(* IEC 61131-3 sources: POC_CAu/, 3 files *)

(* ---- Main 2.0.ST ---- *)
VAR_GLOBAL

//OUTPUT
glob_Pist1 at %Y33.1:BOOL;                                             //pist pod otvorem na vlozeni obrobku
glob_Pist2 at %Y33.0:BOOL;                                             //pist pro lisovani obrobku
glob_Kompresor at %Y33.2:BOOL;                                         //kompresor
glob_MotorStolu at %Y32.5:BOOL;                                        //motor otocneho stolu
glob_DvoucinnyPist1 at %Y32.6:BOOL;                                    //vysunuti dvoucinneho pistu nad dopravnikem
glob_DvoucinnyPist2 at %Y32.7:BOOL;                                    //zasunuti dvoucinneho pistu nad dopravnikem
glob_MotorDopravniku at %Y32.4:BOOL;

//INPUT
glob_Dioda1 at %X100.6:BOOL;                                           //svetelna zavora pod otvorem na vlozeni obrobku
glob_Dioda2 at %X100.0:BOOL;                                           //svetelna zavora na dopravniku
glob_Start_Stop at %X100.7:BOOL;                                       //tlacitko start-stop
glob_TrigStolu at %X100.5:BOOL;                                        //tlacitko, ktere stiskava otoc. stul
glob_tlacitkoPist2 at  %X100.4:BOOL;                                   //tlacitko pod lisem
glob_TlacitkoDopravniku at %X100.1:BOOL;                               //tlacitko u dopravniku

pocetVyrobku: UDINT := 0;
pomSTTrig: USINT := 0;
pomocnaStav:USINT;

glob_KillSwitch:BOOL;

END_VAR

///////////////////////////////////////////////////////////////////////////////////////////////////////////////////////////////////////////////////////////////////////////////////////////////////////

FUNCTION_BLOCK fb_VychoziStav                                          //pocatecni funkce pro nastveni stolu na vychozi pozici

VAR_INPUT
talcitko:BOOL;
END_VAR

VAR_OUTPUT
vystup:BOOL;
END_VAR

VAR
stisknuto:BOOL;
nabezna:R_TRIG;
END_VAR

nabezna(CLK := talcitko,Q => stisknuto);

glob_KillSwitch := glob_KillSwitch XOR stisknuto;

IF glob_TrigStolu = FALSE AND glob_KillSwitch = TRUE THEN
vystup := TRUE;
ELSIF glob_TrigStolu = TRUE THEN
vystup := FALSE;
END_IF;

END_FUNCTION_BLOCK
///////////////////////////////////////////////////////////////////////////////////////////////////////////////////////////////////////////////////////////////////////////////////////////////////////

FUNCTION_BLOCK fb_VypnouLinku                                           //funkce pro vypinani cele linky

VAR_INPUT
talcitko:BOOL;
END_VAR

VAR_OUTPUT
vystup:BOOL;
END_VAR

VAR
stisknuto:BOOL;
nabezna:R_TRIG;
END_VAR

nabezna(CLK := talcitko,Q => stisknuto);

vystup := vystup XOR stisknuto;

IF vystup = FALSE THEN
pomocnaStav:=4;                                                        //obrazuje na display PLC "Pozastaveno"
END_IF;

END_FUNCTION_BLOCK
///////////////////////////////////////////////////////////////////////////////////////////////////////////////////////////////////////////////////////////////////////////////////////////////////////

FUNCTION_BLOCK fb_PozicePist1

VAR_INPUT
dioda1:BOOL;
dioda2:BOOL;
END_VAR

VAR_OUTPUT
vystup1:BOOL;
vystup2:BOOL;
vystup3:BOOL;
END_VAR

VAR
zapnuto:BOOL;
zpozdovac:TON;
END_VAR

zpozdovac1(IN := glob_KillSwitch AND glob_TrigStolu AND NOT dioda1 AND dioda2,PT := T#2s,Q => zapnuto);
vystup1 := zapnuto;
vystup2 := zapnuto;
zpozdovac2(IN := glob_KillSwitch AND dioda1 AND dioda2 AND NOT glob_TlacitkoPist2,PT := T#3s,Q => vystup3);

END_FUNCTION_BLOCK
///////////////////////////////////////////////////////////////////////////////////////////////////////////////////////////////////////////////////////////////////////////////////////////////////////

FUNCTION_BLOCK fb_PoziceLis

VAR_INPUT
tlacitko:BOOL;
END_VAR

VAR_OUTPUT
vystup1:BOOL;
vystup2:BOOL;
vystup3:BOOL;
END_VAR

VAR
zapnuto:BOOL;
zpozdovac:TON;
END_VAR

IF tlacitko = TRUE THEN
zpozdovac(IN := glob_KillSwitch AND glob_TlacitkoPist2,PT := T#5s,Q => zapnuto);
vystup1 := zapnuto;
vystup2 := zapnuto;
vystup3 := zapnuto;
END_IF;

END_FUNCTION_BLOCK
///////////////////////////////////////////////////////////////////////////////////////////////////////////////////////////////////////////////////////////////////////////////////////////////////////

fb_PoziceDopravnik

VAR_INPUT
pist:BOOL;
END_VAR

VAR_OUTPUT
vystup:BOOL;
END_VAR

VAR
vypnut,zapnuto:BOOL;
zpozdovac:TON;
sestupna:F_TRIG;
nabezna:R_TRIG;
END_VAR

sestupna(CLK := pist,Q => vypnut);

IF vypnut = TRUE THEN
glob_MotorStolu := TRUE;
ELSIF glob_TlacitkoDopravniku = TRUE THEN
glob_MotorStolu := FALSE;
END_IF;

zpozdovac(IN := glob_KillSwitch AND glob_TlacitkoDopravniku AND glob_Dioda2,PT := T#1s,Q => vystup);

nabezna(CLK := vystup,Q => zapnuto);

IF zapnuto AND glob_Dioda2 THEN
glob_Kompresor := FALSE;
glob_MotorDopravniku := TRUE;
ELSIF glob_KillSwitch AND NOT glob_Dioda2 THEN
glob_MotorDopravniku := FALSE;
//pocetVyrobku:= pocetVyrobku + 1;
pomocnaStav:=2;                                                        //zobrazuje na display PLC "Odeberte obrobek"
END_IF;

END_FUNCTION_BLOCK
///////////////////////////////////////////////////////////////////////////////////////////////////////////////////////////////////////////////////////////////////////////////////////////////////////

PROGRAM Main

fb_VychoziStav(glob_Start_Stop := tlacitko,vystup := glob_MotorStolu);
fb_VypnouLinku(glob_Start_Stop := tlacitko,vystup := glob_KillSwitch);
fb_PozicePist1(glob_Dioda1 := dioda1,glob_Dioda2 := dioda2,glob_Kompresor := vystup1,glob_Pist1 := vystup2,glob_MotorStolu := vystup3);
fb_PoziceLis(glob_TlacitkoPist2 := tlacitko,glob_Kompresor := vystup1,glob_Pist2 := vystup2,glob_DvoucinnyPist1 := vystup3);
fb_PoziceDopravnik(glob_Pist2 := pist,);

END_PROGRAM

(* ---- prgMain.ST ---- *)
VAR_GLOBAL

//OUTPUT
glob_Pist1 at %Y33.1:BOOL;                                             //pist pod otvorem na vlozeni obrobku
glob_Pist2 at %Y33.0:BOOL;                                             //pist pro lisovani obrobku
glob_Kompresor at %Y33.2:BOOL;                                         //kompresor
glob_MotorStolu at %Y32.5:BOOL;                                        //motor otocneho stolu
glob_DvojcinnyPist1 at %Y32.6:BOOL;                                    //vysunuti dvoucinneho pistu nad dopravnikem
glob_DvojcinnyPist2 at %Y32.7:BOOL;                                    //zasunuti dvoucinneho pistu nad dopravnikem
glob_MotorDopravniku at %Y32.4:BOOL;

//INPUT
glob_Dioda1 at %X100.6:BOOL;                                           //svetelna zavora pod otvorem na vlozeni obrobku
glob_Dioda2 at %X100.0:BOOL;                                           //svetelna zavora na dopravniku
glob_Start_Stop at %X100.7:BOOL;                                       //tlacitko start-stop
glob_TrigStolu at %X100.5:BOOL;                                        //tlacitko, ktere stiskava otoc. stul
glob_tlacitkoPist2 at  %X100.4:BOOL;                                   //tlacitko pod lisem
glob_TlacitkoDopravniku at %X100.1:BOOL;                               //tlacitko u dopravniku

pocetVyrobku: UDINT := 0;
pomocnaStav:USINT;

glob_KillSwitch:BOOL;

END_VAR

///////////////////////////////////////////////////////////////////////////////////////////////////////////////////////////////////////////////////////////////////////////////////////////////////////

FUNCTION_BLOCK fb_VychoziStav

VAR_INPUT
tlacitko:BOOL;
END_VAR

VAR
stisknuto:BOOL;
nabezna:R_TRIG;
END_VAR

nabezna(CLK := tlacitko,Q => stisknuto);
glob_KillSwitch := glob_KillSwitch XOR stisknuto;

IF stisknuto = TRUE THEN
 pomocnaStav:=0;
END_IF;

IF NOT glob_TrigStolu AND glob_KillSwitch THEN
 glob_MotorStolu := TRUE;
ELSIF glob_TrigStolu AND glob_KillSwitch THEN
 glob_MotorStolu := FALSE;
END_IF;

IF glob_KillSwitch = FALSE THEN
 pomocnaStav:=2;
END_IF;

END_FUNCTION_BLOCK
///////////////////////////////////////////////////////////////////////////////////////////////////////////////////////////////////////////////////////////////////////////////////////////////////////

FUNCTION_BLOCK fb_PozicePist1

VAR_INPUT
dioda1:BOOL;
END_VAR

VAR
zapnuto1,zapnuto2,probehlo,pom:BOOL;
zpozdovac1,zpozdovac2:TON;
sestup:F_TRIG;
END_VAR

IF NOT dioda1 THEN
 pomocnaStav:=4;
END_IF;

zpozdovac1(IN := NOT dioda1,PT := T#2s0ms,Q => zapnuto1);

IF zapnuto1 = TRUE THEN
 glob_Kompresor := TRUE;
 glob_Pist1 := TRUE;
 pomocnaStav:=3;
ELSE
 glob_Kompresor := FALSE;
 glob_Pist1 := FALSE;
END_IF;

sestup(CLK := glob_Pist1,Q => probehlo);

if probehlo then;
   pom:=TRUE;
END_IF;

zpozdovac2(IN := pom,PT := T#3s0ms,Q => zapnuto2);

IF zapnuto2 and glob_KillSwitch THEN
   glob_MotorStolu := TRUE;
END_IF;

IF glob_tlacitkoPist2 = TRUE THEN
   glob_MotorStolu := FALSE;
   pom := FALSE;
END_IF;

END_FUNCTION_BLOCK
///////////////////////////////////////////////////////////////////////////////////////////////////////////////////////////////////////////////////////////////////////////////////////////////////////

FUNCTION_BLOCK fb_PoziceLis

VAR_INPUT
tlacitko:BOOL;
END_VAR

VAR
casovac:TP;
sestup:F_TRIG;
zapnuto,probehlo,pom:BOOL;
END_VAR

IF tlacitko = TRUE THEN
 casovac(IN := glob_KillSwitch AND glob_TlacitkoPist2,PT := T#5s0ms,Q => zapnuto);
 glob_Kompresor := zapnuto;
 glob_Pist2 := zapnuto;
 glob_DvojcinnyPist1 := zapnuto;
ELSE
 casovac(IN := FALSE);
END_IF;

sestup(CLK := glob_Pist2,Q => probehlo);

IF probehlo THEN;
 pom := TRUE;
END_IF;

IF pom AND glob_KillSwitch THEN
 glob_MotorStolu := TRUE;
END_IF;

IF glob_TlacitkoDopravniku = TRUE THEN
 glob_MotorStolu := FALSE;
 pom := FALSE;
END_IF;

END_FUNCTION_BLOCK
///////////////////////////////////////////////////////////////////////////////////////////////////////////////////////////////////////////////////////////////////////////////////////////////////////

FUNCTION_BLOCK fb_PoziceDopravnik

VAR_INPUT
tlacitko:BOOL;
END_VAR

VAR
zapnuto,konec,pom:BOOL;
zpozdovac:TON;
nabez:R_TRIG;
END_VAR

IF tlacitko = TRUE THEN
 glob_MotorDopravniku := TRUE;
END_IF;

zpozdovac(IN := glob_KillSwitch AND glob_MotorDopravniku AND glob_Dioda2,PT := T#1s,Q => zapnuto);

IF zapnuto = TRUE THEN
 glob_Kompresor := TRUE;
 glob_DvojcinnyPist2 := TRUE;
END_IF;

nabez(CLK:= NOT glob_Dioda2,Q => konec);

IF glob_Dioda2 = FALSE THEN
 glob_MotorDopravniku := FALSE;
END_IF;

IF konec = TRUE THEN
 pomocnaStav := 1;
 pocetVyrobku := pocetVyrobku + 1;
 pom := TRUE;
END_IF;

IF pom AND glob_Dioda2 THEN
 glob_KillSwitch := FALSE;
 pom := FALSE;
END_IF;

END_FUNCTION_BLOCK
///////////////////////////////////////////////////////////////////////////////////////////////////////////////////////////////////////////////////////////////////////////////////////////////////////

FUNCTION kill : BOOL
         glob_Pist1           :=0;
         glob_Pist2           :=0;
         glob_Kompresor       :=0;
         glob_MotorStolu      :=0;
         glob_DvojcinnyPist1  :=0;
         glob_DvojcinnyPist2  :=0;
         glob_MotorDopravniku :=0;
END_FUNCTION

VAR_GLOBAL
 fb_VS : fb_VychoziStav;
 fb_PP : fb_PozicePist1;
 fb_PL : fb_PoziceLis;
 fb_PD : fb_PoziceDopravnik;
END_VAR

PROGRAM prgMain
fb_VS(tlacitko := glob_Start_Stop);
IF glob_killswitch = TRUE THEN
 fb_PP(dioda1 := glob_Dioda1);
 fb_PL(tlacitko := glob_TlacitkoPist2);
 fb_PD(tlacitko := glob_TlacitkoDopravniku);
ELSE
 kill();
END_IF;

END_PROGRAM

(* ---- OLD_Main.ST ---- *)
VAR_GLOBAL

//OUTPUT
Pist1 at %Y33.1:BOOL;                                                  //pist pod otvorem na vlozeni obrobku
Pist2 at %Y33.0:BOOL;                                                  //pist pro lisovani obrobku
kompr at %Y33.2:BOOL;                                                  //kompresor
MotorStolu at %Y32.5:BOOL;                                             //motor otocneho stolu
DvoucinnyPist1 at %Y32.6:BOOL;                                         //vysunuti dvoucinneho pistu nad dopravnikem
DvoucinnyPist2 at %Y32.7:BOOL;                                         //zasunuti dvoucinneho pistu nad dopravnikem
MotorDopravniku at %Y32.4:BOOL;

//INPUT
Dioda1 at %X100.6:BOOL;                                                //svetelna zavora pod otvorem na vlozeni obrobku
Dioda2 at %X100.0:BOOL;                                                //svetelna zavora na dopravniku
StartStop at %X100.7:BOOL;                                             //tlacitko start-stop
tlacitkoStolu at %X100.5:BOOL;                                         //tlacitko, ktere stiskava otoc. stul
tlacitkoPist2 at  %X100.4:BOOL;                                        //tlacitko pod lisem
tlacitkoDopravniku at %X100.1:BOOL;                                    //tlacitko u dopravniku
pocetVyrobku: UDINT := 0;
pomSTTrig: USINT := 0;
pomocnaStav:USINT;
//prnt at %R1:array[0..79] of USINT;
END_VAR

PROGRAM prgMain

VAR

data:TIME;
nabez1,nebezHotovo:R_TRIG;
sestup1:F_TRIG;
SestupPist2:F_TRIG;
SestuptlacitkoDopravniku:F_TRIG;
Casovac1,Casovac2:TOF;
Zpozdovac1,Zpozdovac2,Zpozdovac3,Zpozdovac4:TON;
pomStart,pomPist1,pomPist2,pomMotorS,pom1,pom3,pom5,pom6,pom7,pom9,pom10,pom11,pom12,pom13,pom14,pom15,pom16,pom17,pom18,pomZap,pomses,pomStop,pomPist1kon,pomZpozdeni,pomHotovo,pomHotovo2,pomHotovo3,pomDonePist1,pomTlacPist2,pomTlacDoublePist3,pomNeco,pomPozastav:BOOL; //pomocne promenne
END_VAR

if pomStart = false then
pomocnaStav:=0;                                                       //zobrazuje na display PLC "Stisknete tlacitko"
pomHotovo2:=false;                                                    //nuluje mezipamet
end_if;

nabez1(CLK:=StartStop,Q=>pom1);

if pom1 then
pomStart:=pomStart xor pom1;                                           //vypinani a zapinani linky
pomocnaStav:=1;                                                        //zobrazuje na display PLC "Vlozte obrobek"
pomSTTrig:=pomSTTrig + 1;
end_if;

(*if (pomSTTrig MOD 2)=0 then;                                         //kazde druhe stisknuti spusti podminku
pomocnaStav:=4;                                                        //obrazuje na display PLC "Pozastaveno"
pomPozastav:=true;                                                     //zaznam o pozastaveni linky
pomSTTrig:=1;
end_if;  *)

if tlacitkoStolu = false and pomStart = true then MotorStolu:= true;   //pocatecni podminka pro nastveni stolu na vychozi pozici
elsif tlacitkoStolu = true then MotorStolu:= false;
end_if;

if not Dioda1 and pomStart and Dioda2 then                             //podminka pro spusteni Pist1, kdyz je vlozen obrobek a je odebrán obrobek z dopravníku
pom10:= true;                                                          //pomocna pro zaznamenani aktivace casovace se zpozdenim 2s

elsif Pist1 = true then
//pomocnaStav:=0;
pom7:= true;                                                           //pomocna pro zaznamenani aktivace Pist1
pomDonePist1:=true;

elsif pom10 and pom7 and pomStart then                                 //pokud probehl casovac (Zpozdovac1) se spozdenim 2s a Pist1 se vysunul
pomMotorS:= not tlacitkoPist2 and Dioda1 and pomStart;                 //pomocna pro spusteni casovace Zpozdovac2
MotorStolu:= pom5;                                                     //zapinani motoru otocneho stolu
pom12:= true;                                                          //zaznamenani o probehlem otoceni stolu
end_if;

Zpozdovac1(IN:= not Dioda1 and pomStart and Dioda2 and tlacitkoStolu,PT:= T#2s,Q=>pom3,ET=>data);//zpozdeny start 2s
kompr:= pom3;                                                          //zapnuti kompresoru
Pist1:= kompr;                                                         //zapnuti pneumatickeho lisu (Pist1), ktery vysune obrobek na otocny stul

if Pist1 = true then                                                   //blbuvzdornost pri startu Pistu2
pomPist1kon:= true;                                                    //zaznamenani akce do pameti
end_if;

Zpozdovac2(IN:= pomMotorS,PT:= T#3s,Q=>pom5,ET=>data);                 //zpozdeny start 3s
if pom5 = true then
pomZpozdeni:= true;
end_if;

if tlacitkoPist2 and pomStart and pomPist1kon then                     //pokud je stisknuto tlacitkoStolu, motor otoc. stolu se zastavi
kompr:= not pom9;                                                      //zapnuti kompresoru
Pist2:= not pom9;                                                      //zapnuti pneumatickeho lisu (Pist2), ktery stalci obrobek
DvoucinnyPist1:= not pom9;                                             //zapnuti dvoucinneho pneumatickeho lisu (DvoucinnyPist1)
DvoucinnyPist2:=false;                                                 //nulovani dvoucinneho pneumatickeho lisu (DvoucinnyPist2)
pom11:= true;                                                          //zaznamenani o probehlem spusteni pistu (Pist2)
pom10:=false;                                                          //blokace motoru otoc. stolu
pom7:=false;                                                           //blokace motoru otoc. stolu
pomTlacPist2:=true;                                                    //zaznamenani akce do pameti
end_if;

Zpozdovac3(IN:= tlacitkoPist2 and pomStart,PT:= T#5s,Q=>pom9,ET=>data);//zpozdene zapnuti 5s

SestupPist2(clk:=Pist2,Q=>pom13);                                      //zaznamenani sestupne hrany, kdyz Pist2 se vypne

if pom13 = true then                                                   //pokud byl Pist2 vypnut spusti se podminka
pom14:= true;
end_if;

if pom11 and pom14 and not tlacitkoDopravniku and pomStart then        //pokud byl Pist2 spusten a nasledne vypnut spusti se podminka pro zapnuti otoc. stolu do doby nez se dotkne tlacitkoDopravniku
MotorStolu:=true;

elsif pom17 and pomStart and Dioda2 then                               //zda-li obrobek stiskl tlacitoStolu
kompr:=true;
DvoucinnyPist1:=false;                                                 //zapnuti kompresoru
DvoucinnyPist2:= true;                                                 //zapnuti dvoucinneho pneumatickeho lisu (DvoucinnyPist2)
pomTlacDoublePist3:=true;                                              //zaznamenani akce do pameti
pom11:=false;
pom14:=false;                                                          //blokace predchozi podminky, aby se znovu nespustil otoc. stul, kdyz obrobek uz netlaci na tlacitkoStolu
pom16:=true;                                                           //zaznam o probehle akci
end_if;

Zpozdovac4(IN:= tlacitkoDopravniku,PT:= T#1s,Q=>pom15,ET=>data);       //ceka 1s na presun obrobku na dostavnik
pom17:=pom15;

if pom16 and Dioda2 and pomStart then                                  //spusti motorDopravniku do doby, kdy obrobek nedojede do svetelnou zavorou (Dioda2)
MotorDopravniku:= true;

SestuptlacitkoDopravniku(clk:=tlacitkoDopravniku,Q=>pom18);            //zaznam sestupne hrany

elsif pom18 then                                                       //pote co se obrobek odebere na pas, vypne kompresor
kompr:=false;

elsif not Dioda2 then                                                  //kdyz obrobek stoji ve svetelne zavore, tak vypina motor dopravniku a kompresor
MotorDopravniku:= false;
pom16:=false;
pom6:=pomHotovo;
end_if;

nebezHotovo(clk:= not Dioda2,Q=>pomHotovo);                            //1 zaznam o vyskytu obrobku ve druhe svetelne zavore (Dioada2)

if pom6 and pomTlacDoublePist3 and pomTlacPist2 and pomDonePist1 and not Dioda2 and not pomPozastav then
pocetVyrobku:=pocetVyrobku+1;                                          //pripocteni +1 k obrobenych obrobku
pomocnaStav:=2;                                                        //zobrazuje na display PLC "Odeberte obrobek"
pomHotovo2:=true;
end_if;

*(if pomStart and pomPozastav then
pomocnaStav:=2;
pomHotovo2:=true;
end_if;*)

if pomHotovo2 and Dioda2 then                                          //nulovani pameti
pomStart:=false;
pomTlacDoublePist3:=false;
pomTlacPist2:=false;
pomDonePist1:=false;
pomHotovo3:=true;
pomPozastav:=false;
end_if;

(*if pomHotovo3 and Dioda1 then
pomocnaStav:=1;
pomHotovo2:=false;
end_if;*)

if pomStart and not Dioda1 then                                        //zobrazuje na display PLC "_"
pomocnaStav:=3;
end_if;

(*if pom6 = true then
pomStart:=false;
pomocnaStav:=0;
end_if;*)

END_PROGRAM
